// TIA Portal V17 export
// export: Created 2024-12-18T11:14:19.8547058Z, ExportSetting WithDefaults, DisplayName Totally Integrated Automation Portal, DisplayVersion V17 Update 6, DisplayName TIA Portal Openness, DisplayVersion V17 Update 6, DisplayName TIA Portal Version Control Interface, DisplayVersion V17, DisplayName SINAMICS Startdrive Advanced, DisplayVersion V17 SP1, DisplayName SINAMICS Startdrive G130, G150, S120, S150, SINAMICS MV, S210, DisplayVersion V17 SP1, DisplayName SINAMICS Startdrive G110M, G120, G120C, G120D, G120P, G115D, DisplayVersion V17 SP1, DisplayName STEP 7 Professional, DisplayVersion V17 Update 6, DisplayName SINUMERIK ONE STEP 7 Toolbox, DisplayVersion V17 Update 2, DisplayName SINUMERIK 840D sl STEP 7 Toolbox, DisplayVersion V17 Update 2, DisplayName STEP 7 Safety, DisplayVersion V17 Update 6, DisplayName WinCC Advanced / Unified PC, DisplayVersion V17 Update 6
TYPE "UDT_Test"
// stored: IsFailsafeCompliant false
   STRUCT
      "Bool" : Bool;
      int1 : Int;
      int2 : Int;
   END_STRUCT;
END_TYPE
